FUNCTION flip_int : ARRAY[0..3] OF BYTE
VAR_INPUT
	valor_real : INT;
END_VAR

VAR
		valor_byte :  ARRAY[0..3] OF BYTE;
		valor_flip : ARRAY[0..3] OF BYTE;
		pByteIn1, pByteIn2, pByteIn3, pByteIn4: POINTER TO BYTE;
		

		
END_VAR


//direcciones
pByteIn1 := ADR(valor_real);
pByteIn2 := ADR(valor_real) + SIZEOF(BYTE);
pByteIn3 := ADR(valor_real) + 2 * SIZEOF(BYTE);
pByteIn4 := ADR(valor_real) + 3 * SIZEOF(BYTE);



valor_byte[0] := pByteIn1^;
valor_byte[1] := pByteIn2^ ;
valor_byte[2] := pByteIn3^ ;
valor_byte[3] := pByteIn4^ ;

valor_flip[0] := valor_byte[3];
valor_flip[1] := valor_byte[2];
valor_flip[2] := valor_byte[1];
valor_flip[3] := valor_byte[0];


flip_int := valor_flip;

END_FUNCTION

(* stored: Version 1.1.0.1, ProductVersion 3.1.4024.4
   POU flip_int: Id {5218a208-f11c-4cfe-ad06-5dd5a12c4f12}, SpecialFunc None *)
